% RSLogix 500 project BIO_DIESEL_BAK001.RSS, saved by version 8.30.00.16 %
PROJECT "UNTITLED"    % processor: Bul.1763 MicroLogix 1100 Series A %

PROGRAM FILES
  LAD 2 "MAIN"  15 rungs
  LAD 3 "PID"  4 rungs

DATA FILES
  O0 OUTPUT  4 elements
  I1 INPUT  6 elements
  S2 STATUS  66 elements
  B3 BINARY  1 elements
  T4 TIMER  3 elements
  C5 COUNTER  1 elements
  R6 CONTROL  1 elements
  N7 INTEGER  6 elements
  F8 FLOAT  1 elements
  PD9 PID_09  1 elements

LADDER 2 "MAIN"
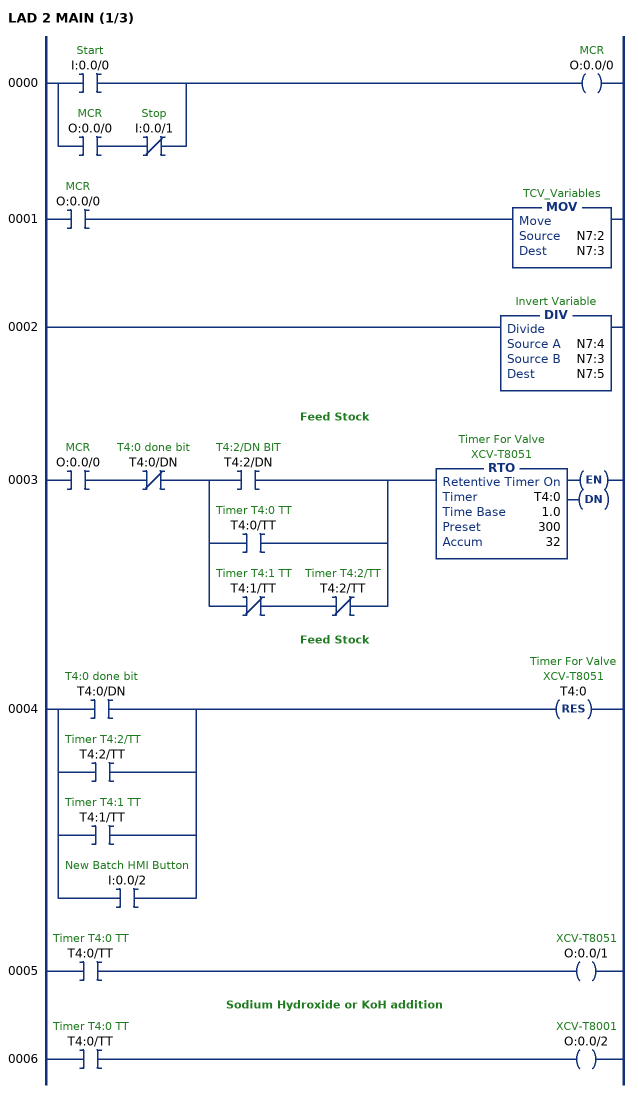
% Rung: 0 %
SOR BST XIC I:0.0/0 NXB XIC O:0.0/0 XIO I:0.0/1 BND OTE O:0.0/0 EOR
%   I:0.0/0  "Start" %
%   O:0.0/0  "MCR" %
%   I:0.0/1  "Stop" %
% Rung: 1 %
SOR XIC O:0.0/0 MOV N7:2 N7:3 EOR
%   O:0.0/0  "MCR" %
%   N7:2  N7 %
%   N7:3  "TCV_Variables" %
% Rung: 2 %
SOR DIV N7:4 N7:3 N7:5 EOR
%   N7:4  "Invert TCV Variable" %
%   N7:3  "TCV_Variables" %
%   N7:5  "Invert Variable" %
% Rung: 3 %
% TITLE: Feed Stock %
SOR XIC O:0.0/0 XIO T4:0/DN BST XIC T4:2/DN NXB XIC T4:0/TT NXB XIO T4:1/TT XIO T4:2/TT BND RTO T4:0 1.0 300 32 EOR
%   O:0.0/0  "MCR" %
%   T4:0/DN  "T4:0 done bit" %
%   T4:2/DN  "T4:2/DN BIT" %
%   T4:0/TT  "Timer T4:0 TT" %
%   T4:1/TT  "Timer T4:1 TT" %
%   T4:2/TT  "Timer T4:2/TT" %
%   T4:0  "Timer For Valve XCV-T8051" %
% Rung: 4 %
% TITLE: Feed Stock %
SOR BST XIC T4:0/DN NXB XIC T4:2/TT NXB XIC T4:1/TT NXB XIC I:0.0/2 BND RES T4:0 EOR
%   T4:0/DN  "T4:0 done bit" %
%   T4:2/TT  "Timer T4:2/TT" %
%   T4:1/TT  "Timer T4:1 TT" %
%   I:0.0/2  "New Batch HMI Button" %
%   T4:0  "Timer For Valve XCV-T8051" %
% Rung: 5 %
SOR XIC T4:0/TT OTE O:0.0/1 EOR
%   T4:0/TT  "Timer T4:0 TT" %
%   O:0.0/1  "XCV-T8051" %
% Rung: 6 %
% TITLE: Sodium Hydroxide or KoH addition %
SOR XIC T4:0/TT OTE O:0.0/2 EOR
%   T4:0/TT  "Timer T4:0 TT" %
%   O:0.0/2  "XCV-T8001" %

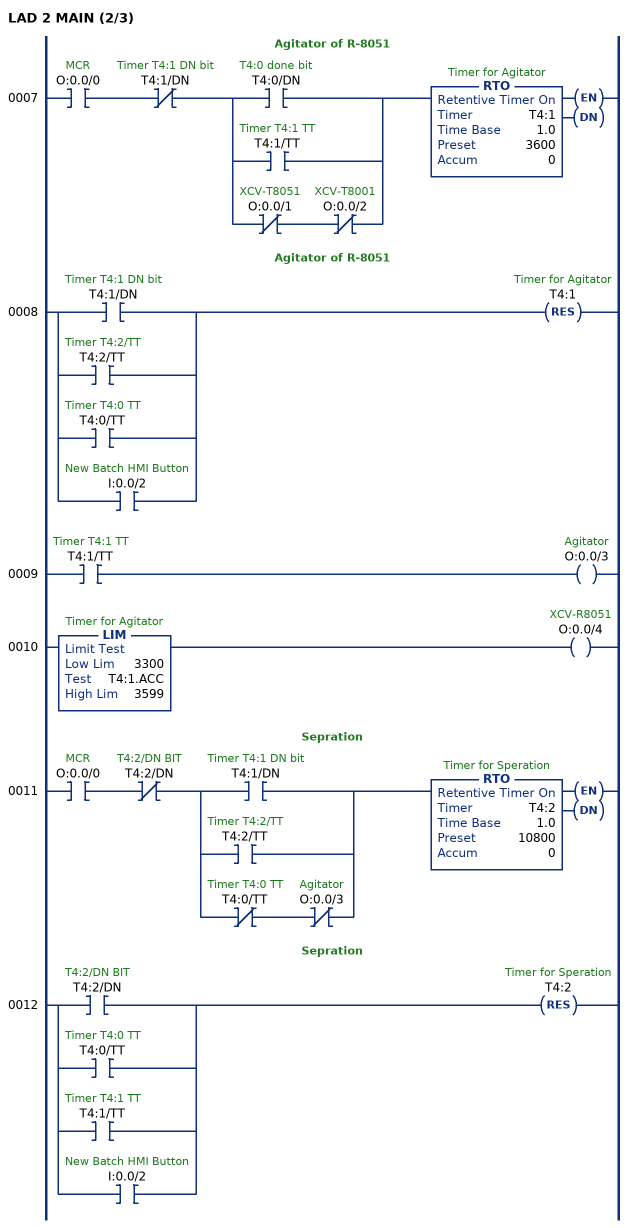
% Rung: 7 %
% TITLE: Agitator of R-8051 %
SOR XIC O:0.0/0 XIO T4:1/DN BST XIC T4:0/DN NXB XIC T4:1/TT NXB XIO O:0.0/1 XIO O:0.0/2 BND RTO T4:1 1.0 3600 0 EOR
%   O:0.0/0  "MCR" %
%   T4:1/DN  "Timer T4:1 DN bit" %
%   T4:0/DN  "T4:0 done bit" %
%   T4:1/TT  "Timer T4:1 TT" %
%   O:0.0/1  "XCV-T8051" %
%   O:0.0/2  "XCV-T8001" %
%   T4:1  "Timer for Agitator" %
% Rung: 8 %
% TITLE: Agitator of R-8051 %
SOR BST XIC T4:1/DN NXB XIC T4:2/TT NXB XIC T4:0/TT NXB XIC I:0.0/2 BND RES T4:1 EOR
%   T4:1/DN  "Timer T4:1 DN bit" %
%   T4:2/TT  "Timer T4:2/TT" %
%   T4:0/TT  "Timer T4:0 TT" %
%   I:0.0/2  "New Batch HMI Button" %
%   T4:1  "Timer for Agitator" %
% Rung: 9 %
SOR XIC T4:1/TT OTE O:0.0/3 EOR
%   T4:1/TT  "Timer T4:1 TT" %
%   O:0.0/3  "Agitator" %
% Rung: 10 %
SOR LIM 3300 T4:1.ACC 3599 OTE O:0.0/4 EOR
%   T4:1  "Timer for Agitator" %
%   O:0.0/4  "XCV-R8051" %
% Rung: 11 %
% TITLE: Sepration %
SOR XIC O:0.0/0 XIO T4:2/DN BST XIC T4:1/DN NXB XIC T4:2/TT NXB XIO T4:0/TT XIO O:0.0/3 BND RTO T4:2 1.0 10800 0 EOR
%   O:0.0/0  "MCR" %
%   T4:2/DN  "T4:2/DN BIT" %
%   T4:1/DN  "Timer T4:1 DN bit" %
%   T4:2/TT  "Timer T4:2/TT" %
%   T4:0/TT  "Timer T4:0 TT" %
%   O:0.0/3  "Agitator" %
%   T4:2  "Timer for Speration" %
% Rung: 12 %
% TITLE: Sepration %
SOR BST XIC T4:2/DN NXB XIC T4:0/TT NXB XIC T4:1/TT NXB XIC I:0.0/2 BND RES T4:2 EOR
%   T4:2/DN  "T4:2/DN BIT" %
%   T4:0/TT  "Timer T4:0 TT" %
%   T4:1/TT  "Timer T4:1 TT" %
%   I:0.0/2  "New Batch HMI Button" %
%   T4:2  "Timer for Speration" %

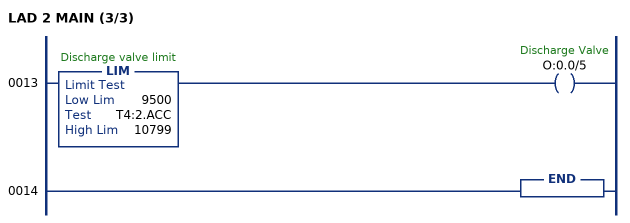
% Rung: 13 %
SOR LIM 9500 T4:2.ACC 10799 OTE O:0.0/5 EOR
%   T4:2.ACC  "Discharge valve limit" %
%   O:0.0/5  "Discharge Valve" %
% Rung: 14 %
SOR END EOR

LADDER 3 "PID"
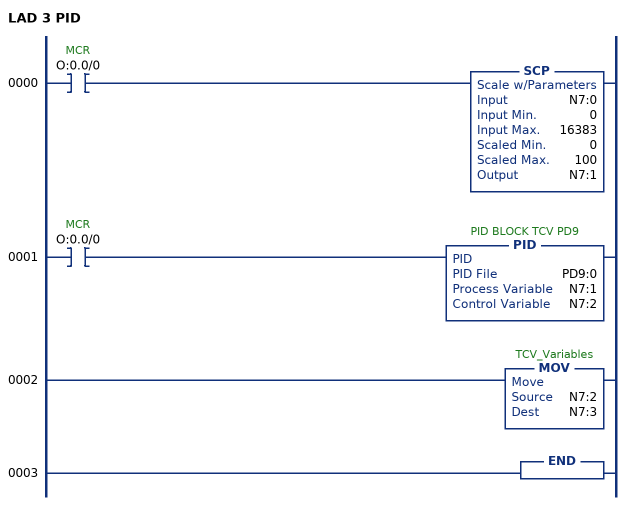
% Rung: 0 %
SOR XIC O:0.0/0 SCP N7:0 0 16383 0 100 N7:1 EOR
%   O:0.0/0  "MCR" %
%   N7:0  "Temperature Sensor" %
% Rung: 1 %
SOR XIC O:0.0/0 PID PD9:0 N7:1 N7:2 EOR
%   O:0.0/0  "MCR" %
%   PD9:0  PD9  "PID BLOCK TCV" %
%   N7:2  N7 %
% Rung: 2 %
SOR MOV N7:2 N7:3 EOR
%   N7:2  N7 %
%   N7:3  "TCV_Variables" %
% Rung: 3 %
SOR END EOR

DATA TABLE (non-zero values as saved)
DATA T4
% .PRE .ACC %
% T4:0 % 300 32
% T4:1 % 3600 0
% T4:2 % 10800 0
DATA N7
% N7:0 % 9010 55 60 60 1 0
